// TIA Portal V17 export
// export: Created 2025-03-10T12:16:55.6331284Z, ExportSetting WithDefaults, DisplayName Totally Integrated Automation Portal, DisplayVersion V17 Update 8, DisplayName TIA Portal Openness, DisplayVersion V17 Update 8, DisplayName TIA Portal Version Control Interface, DisplayVersion V17, DisplayName SINAMICS Startdrive Advanced, DisplayVersion V17 SP2, DisplayName SINAMICS Startdrive G110M, G120, G120C, G120D, G120P, G115D, DisplayVersion V17 SP2, DisplayName SINAMICS Startdrive G130, G150, S120, S150, SINAMICS MV, S210, DisplayVersion V17 SP2, DisplayName STEP 7 Professional, DisplayVersion V17 Update 8, DisplayName SINUMERIK ONE STEP 7 Toolbox, DisplayVersion V17 Update 12, DisplayName SINUMERIK 840D sl STEP 7 Toolbox, DisplayVersion V17 Update 12, DisplayName STEP 7 Safety, DisplayVersion V17 Update 6, DisplayName WinCC Advanced, DisplayVersion V17 Update 8
FUNCTION "FC6691_UNIT_01_STA_3_AXIAL_LOCATOR" : Void   // FC6691, LAD
{ S7_Optimized_Access := 'TRUE' }
VERSION : 0.1
// stored: AutoNumber false, IsIECCheckEnabled false, SetENOAutomatically false, UDAEnableTagReadback false
BEGIN

REGION Network 1: CALL FB6500 UNIT 01 STATION 3 AXIAL LOCATOR
   // 2#0000_0001 OPTIONS 0 BIT 0 ADVANCED INPUT 1 OPTION
   // 2#0000_0010 OPTIONS 0 BIT 1 ADVANCED INPUT 2 OPTION
   // 2#0000_0100 OPTIONS 0 BIT 2 ADVANCED INPUT 3 OPTION
   // 2#0000_1000 OPTIONS 0 BIT 3 ADVANCED INPUT 4 OPTION
   // 2#0001_0000 OPTIONS 0 BIT 4 RETURNED INPUT 1 OPTION
   // 2#0010_0000 OPTIONS 0 BIT 5 RETURNED INPUT 2 OPTION
   // 2#0100_0000 OPTIONS 0 BIT 6 RETURNED INPUT 3 OPTION
   // 2#1000_0000 OPTIONS 0 BIT 7 RETURNED INPUT 4 OPTION
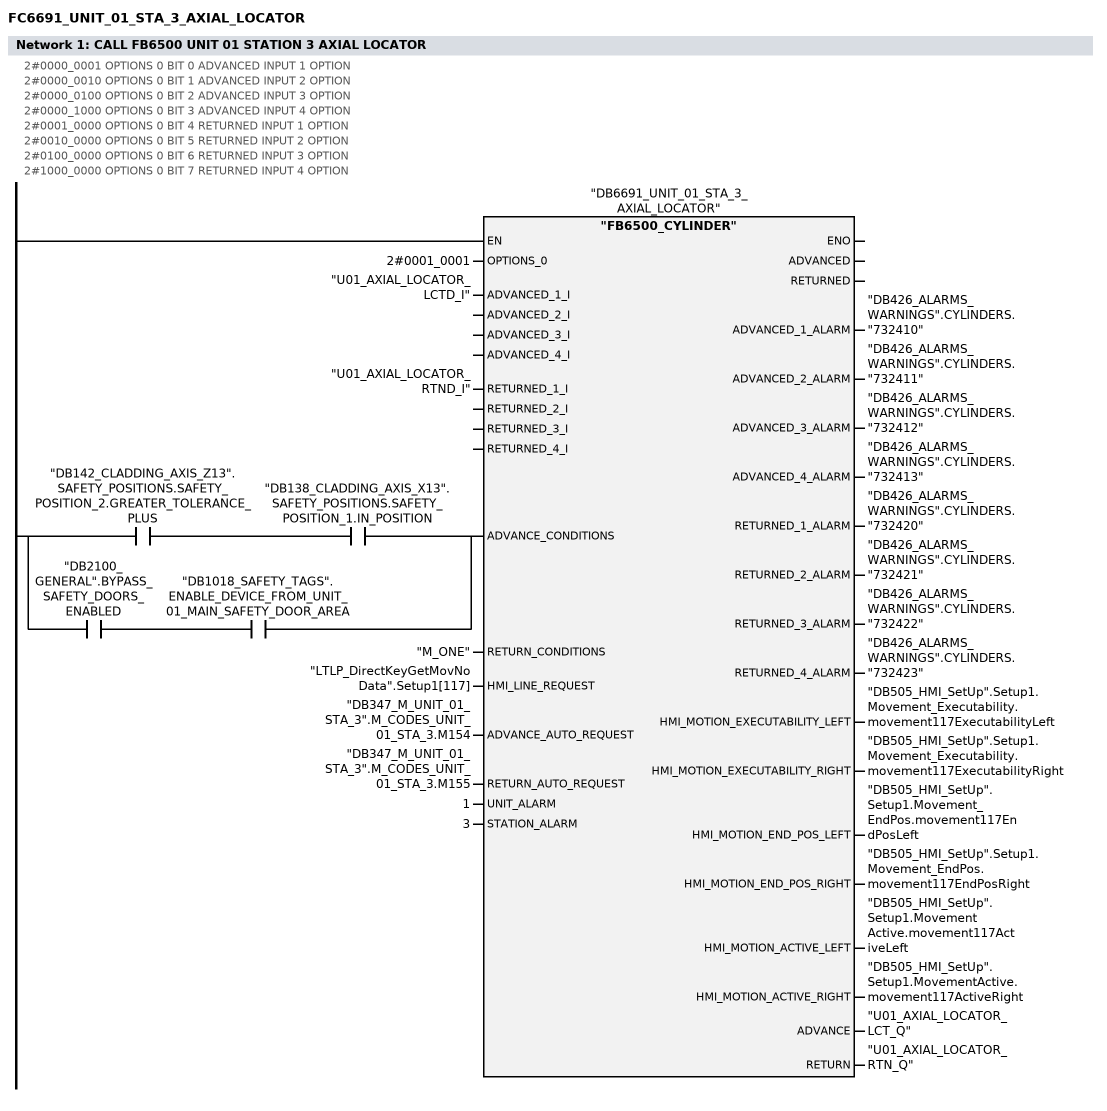
   RUNG wire#powerrail
      "DB6691_UNIT_01_STA_3_AXIAL_LOCATOR"(ADVANCE_CONDITIONS := wire#w1, OPTIONS_0 := 2#0001_0001, ADVANCED_1_I := "U01_AXIAL_LOCATOR_LCTD_I", ADVANCED_2_I :=, ADVANCED_3_I :=, ADVANCED_4_I :=, RETURNED_1_I := "U01_AXIAL_LOCATOR_RTND_I", RETURNED_2_I :=, RETURNED_3_I :=, RETURNED_4_I :=, RETURN_CONDITIONS := "M_ONE", HMI_LINE_REQUEST := "LTLP_DirectKeyGetMovNoData".Setup1[117], ADVANCE_AUTO_REQUEST := "DB347_M_UNIT_01_STA_3".M_CODES_UNIT_01_STA_3.M154, RETURN_AUTO_REQUEST := "DB347_M_UNIT_01_STA_3".M_CODES_UNIT_01_STA_3.M155, UNIT_ALARM := 1, STATION_ALARM := 3, ADVANCED =>, RETURNED =>, ADVANCED_1_ALARM => "DB426_ALARMS_WARNINGS".CYLINDERS."732410", ADVANCED_2_ALARM => "DB426_ALARMS_WARNINGS".CYLINDERS."732411", ADVANCED_3_ALARM => "DB426_ALARMS_WARNINGS".CYLINDERS."732412", ADVANCED_4_ALARM => "DB426_ALARMS_WARNINGS".CYLINDERS."732413", RETURNED_1_ALARM => "DB426_ALARMS_WARNINGS".CYLINDERS."732420", RETURNED_2_ALARM => "DB426_ALARMS_WARNINGS".CYLINDERS."732421", RETURNED_3_ALARM => "DB426_ALARMS_WARNINGS".CYLINDERS."732422", RETURNED_4_ALARM => "DB426_ALARMS_WARNINGS".CYLINDERS."732423", HMI_MOTION_EXECUTABILITY_LEFT => "DB505_HMI_SetUp".Setup1.Movement_Executability.movement117ExecutabilityLeft, HMI_MOTION_EXECUTABILITY_RIGHT => "DB505_HMI_SetUp".Setup1.Movement_Executability.movement117ExecutabilityRight, HMI_MOTION_END_POS_LEFT => "DB505_HMI_SetUp".Setup1.Movement_EndPos.movement117EndPosLeft, HMI_MOTION_END_POS_RIGHT => "DB505_HMI_SetUp".Setup1.Movement_EndPos.movement117EndPosRight, HMI_MOTION_ACTIVE_LEFT => "DB505_HMI_SetUp".Setup1.MovementActive.movement117ActiveLeft, HMI_MOTION_ACTIVE_RIGHT => "DB505_HMI_SetUp".Setup1.MovementActive.movement117ActiveRight, ADVANCE => "U01_AXIAL_LOCATOR_LCT_Q", "RETURN" => "U01_AXIAL_LOCATOR_RTN_Q")
   END_RUNG
   RUNG wire#powerrail
      Contact( "DB142_CLADDING_AXIS_Z13".SAFETY_POSITIONS.SAFETY_POSITION_2.GREATER_TOLERANCE_PLUS )
      Contact( "DB138_CLADDING_AXIS_X13".SAFETY_POSITIONS.SAFETY_POSITION_1.IN_POSITION )
   END_RUNG wire#w1
   RUNG wire#powerrail
      Contact( "DB2100_GENERAL".BYPASS_SAFETY_DOORS_ENABLED )
      Contact( "DB1018_SAFETY_TAGS".ENABLE_DEVICE_FROM_UNIT_01_MAIN_SAFETY_DOOR_AREA )
   END_RUNG wire#w1
   // the same network as SCL:
   "DB6691_UNIT_01_STA_3_AXIAL_LOCATOR"(OPTIONS_0 := 2#0001_0001,   // "FB6500_CYLINDER"
                           ADVANCED_1_I := "U01_AXIAL_LOCATOR_LCTD_I",
                           RETURNED_1_I := "U01_AXIAL_LOCATOR_RTND_I",
                           ADVANCE_CONDITIONS := ("DB142_CLADDING_AXIS_Z13".SAFETY_POSITIONS.SAFETY_POSITION_2.GREATER_TOLERANCE_PLUS AND "DB138_CLADDING_AXIS_X13".SAFETY_POSITIONS.SAFETY_POSITION_1.IN_POSITION) OR ("DB2100_GENERAL".BYPASS_SAFETY_DOORS_ENABLED AND "DB1018_SAFETY_TAGS".ENABLE_DEVICE_FROM_UNIT_01_MAIN_SAFETY_DOOR_AREA),
                           RETURN_CONDITIONS := "M_ONE",
                           HMI_LINE_REQUEST := "LTLP_DirectKeyGetMovNoData".Setup1[117],
                           ADVANCE_AUTO_REQUEST := "DB347_M_UNIT_01_STA_3".M_CODES_UNIT_01_STA_3.M154,
                           RETURN_AUTO_REQUEST := "DB347_M_UNIT_01_STA_3".M_CODES_UNIT_01_STA_3.M155,
                           UNIT_ALARM := 1,
                           STATION_ALARM := 3,
                           ADVANCED_1_ALARM => "DB426_ALARMS_WARNINGS".CYLINDERS."732410",
                           ADVANCED_2_ALARM => "DB426_ALARMS_WARNINGS".CYLINDERS."732411",
                           ADVANCED_3_ALARM => "DB426_ALARMS_WARNINGS".CYLINDERS."732412",
                           ADVANCED_4_ALARM => "DB426_ALARMS_WARNINGS".CYLINDERS."732413",
                           RETURNED_1_ALARM => "DB426_ALARMS_WARNINGS".CYLINDERS."732420",
                           RETURNED_2_ALARM => "DB426_ALARMS_WARNINGS".CYLINDERS."732421",
                           RETURNED_3_ALARM => "DB426_ALARMS_WARNINGS".CYLINDERS."732422",
                           RETURNED_4_ALARM => "DB426_ALARMS_WARNINGS".CYLINDERS."732423",
                           HMI_MOTION_EXECUTABILITY_LEFT => "DB505_HMI_SetUp".Setup1.Movement_Executability.movement117ExecutabilityLeft,
                           HMI_MOTION_EXECUTABILITY_RIGHT => "DB505_HMI_SetUp".Setup1.Movement_Executability.movement117ExecutabilityRight,
                           HMI_MOTION_END_POS_LEFT => "DB505_HMI_SetUp".Setup1.Movement_EndPos.movement117EndPosLeft,
                           HMI_MOTION_END_POS_RIGHT => "DB505_HMI_SetUp".Setup1.Movement_EndPos.movement117EndPosRight,
                           HMI_MOTION_ACTIVE_LEFT => "DB505_HMI_SetUp".Setup1.MovementActive.movement117ActiveLeft,
                           HMI_MOTION_ACTIVE_RIGHT => "DB505_HMI_SetUp".Setup1.MovementActive.movement117ActiveRight,
                           ADVANCE => "U01_AXIAL_LOCATOR_LCT_Q",
                           "RETURN" => "U01_AXIAL_LOCATOR_RTN_Q");
END_REGION
END_FUNCTION
